{attribute 'GeneratedUsingTerminal: EK1122-0000-0018'}
{attribute addProperty BoxType "EK1122-0000-0018"}
{attribute addProperty Id "Beckhoff_EPP2xxxsub_EK1100EK1100_AB5A94672A_0001_EPP2008_0001_0016EPP2008_D86968E311A_0002_EPP2008_0001_0017EPP2008_D86968E311A_0003_EPP2008_0001_0018EPP2008_D86968E311A_0004_EPP2008_0002_0016EPP2008_D86968E311A_0005_EPP2008_0002_0017EPP2008_D86968E311A_0006_EPP2008_0002_0018EPP2008_D86968E311A_0007_EPP2008_0022_0016EPP2008_D86968E311A_0008_EPP2028_0001_0016EPP2028_D86968E311A_0009_EPP2028_0001_0017EPP2028_D86968E311A_0010_EPP2028_0002_0016EPP2028_D86968E311A_0011_EPP2028_0002_0017EPP2028_D86968E311A_0012_EPP2038_0001_0016EPP2038_0667821720A_0013_EPP2038_0002_0016EPP2038_0667821720A_0014_EPP2304_0061_0016EPP2304_2989DBB88A_0015_EPP2304_0061_0017EPP2304_2989DBB88A_0016_EPP2304_0061_0018EPP2304_2989DBB88A_0017_EPP2308_0001_0016EPP2308_CC30ABA712A_0018_EPP2308_0001_0017EPP2308_CC30ABA712A_0019_EPP2308_0001_0018EPP2308_CC30ABA712A_0020_EPP2308_0002_0016EPP2308_CC30ABA712A_0021_EPP2308_0002_0017EPP2308_CC30ABA712A_0022_EPP2308_0002_0018EPP2308_CC30ABA712A_0023_EPP2316_0003_0016EPP2316_ACB55CD744A_0024_EPP2316_0003_0017EPP2316_ACB55CD744A_0025_EPP2316_0003_0018EPP2316_B4F7513944A_0026_EPP2316_0008_0016EPP2316_ACB55CD744A_0027_EPP2316_0008_0017EPP2316_ACB55CD744A_0028_EPP2316_0008_0018EPP2316_B4F7513944A_0029_EPP2318_0001_0016EPP2318_CC30ABA712A_0030_EPP2318_0001_0017EPP2318_CC30ABA712A_0031_EPP2318_0001_0018EPP2318_CC30ABA712A_0032_EPP2318_0002_0016EPP2318_CC30ABA712A_0033_EPP2318_0002_0017EPP2318_CC30ABA712A_0034_EPP2318_0002_0018EPP2318_CC30ABA712A_0035_EPP2328_0001_0016EPP2328_CC30ABA712A_0036_EPP2328_0001_0017EPP2328_CC30ABA712A_0037_EPP2328_0001_0018EPP2328_CC30ABA712A_0038_EPP2328_0002_0016EPP2328_CC30ABA712A_0039_EPP2328_0002_0017EPP2328_CC30ABA712A_0040_EPP2328_0002_0018EPP2328_CC30ABA712A_0041_EPP2334_0061_0016EPP2334_CC30ABA712A_0042_EPP2334_0061_0017EPP2334_CC30ABA712A_0043_EPP2334_0061_0018EPP2334_CC30ABA712A_0044_EPP2334_0061_0019EPP2334_CC30ABA712A_0045_EPP2338_0001_0016EPP2338_B9F455E920A_0046_EPP2338_0001_0017EPP2338_B9F455E920A_0047_EPP2338_0001_0018EPP2338_B9F455E920A_0048_EPP2338_0002_0016EPP2338_B9F455E920A_0049_EPP2338_0002_0017EPP2338_B9F455E920A_0050_EPP2338_0002_0018EPP2338_B9F455E920A_0051_EPP2338_1001_0017EPP2338_B9F455E920A_0052_EPP2338_1001_0018EPP2338_B9F455E920A_0053_EPP2338_1001_0019EPP2338_B9F455E920A_0054_EPP2338_1002_0017EPP2338_B9F455E920A_0055_EPP2338_1002_0018EPP2338_B9F455E920A_0056_EPP2338_1002_0019EPP2338_B9F455E920A_0057_EPP2339_0003_0016EPP2339_509ECB0F50A_0058_EPP2339_0021_0016EPP2339_618EB00436A_0059_EPP2339_0021_0017EPP2339_0ADD710F36A_0060_EPP2339_0021_0018EPP2339_0ADD710F36A_0061_EPP2339_0022_0016EPP2339_618EB00436A_0062_EPP2339_0022_0017EPP2339_0ADD710F36A_0063_EPP2339_0022_0018EPP2339_0ADD710F36A_0064_EPP2349_0021_0016EPP2349_618EB00436A_0065_EPP2349_0021_0017EPP2349_0ADD710F36A_0066_EPP2349_0021_0018EPP2349_0ADD710F36A_0067_EPP2349_0022_0016EPP2349_618EB00436A_0068_EPP2349_0022_0017EPP2349_0ADD710F36A_0069_EPP2349_0022_0018EPP2349_0ADD710F36A_0070_EPP2624_0002_0016EPP2624_15DDA43F7A_0071_EPP2809_0021_0016EPP2809_E4096AA219A_0072_EPP2809_0022_0016EPP2809_E4096AA219A_0073_EPP2816_0004_0016EPP2816_C5A667B351A_0074_EPP2816_0004_0017EPP2816_C5A667B351A_0075_EPP2816_0008_0016EPP2816_2E3F94AC51A_0076_EPP2816_0008_0017EPP2816_2E3F94AC51A_0077_EPP2816_0008_0018EPP2816_2E3F94AC51A_0078_EPP2816_0010_0016EPP2816_2E3F94AC51A_0079_EPP2816_0010_0017EPP2816_2E3F94AC51A_0080_EPP2816_0010_0018EPP2816_2E3F94AC51A_0081_EPP2817_0008_0016EPP2817_1E85A59C70A_0082_EPP2817_0008_0017EPP2817_1E85A59C70A_0083_EPP2817_0008_0018EPP2817_1E85A59C70"}
{attribute addProperty CRC "1991220122"}
{attribute addProperty Size "2100"}
TYPE Beckhoff_EPP2xxxEK1122_76AF9B9A EXTENDS EK1122_AB5A9467 :
STRUCT
	{attribute addProperty Name "Beckhoff_EPP2xxxsub_EK1100"}
	Beckhoff_EPP2xxxsub_EK1100 : EK1100_AB5A9467;
	{attribute addProperty Name "A_0001_EPP2008_0001_0016"}
	A_0001_EPP2008_0001_0016 : EPP2008_D86968E3;
	{attribute addProperty Name "A_0002_EPP2008_0001_0017"}
	A_0002_EPP2008_0001_0017 : EPP2008_D86968E3;
	{attribute addProperty Name "A_0003_EPP2008_0001_0018"}
	A_0003_EPP2008_0001_0018 : EPP2008_D86968E3;
	{attribute addProperty Name "A_0004_EPP2008_0002_0016"}
	A_0004_EPP2008_0002_0016 : EPP2008_D86968E3;
	{attribute addProperty Name "A_0005_EPP2008_0002_0017"}
	A_0005_EPP2008_0002_0017 : EPP2008_D86968E3;
	{attribute addProperty Name "A_0006_EPP2008_0002_0018"}
	A_0006_EPP2008_0002_0018 : EPP2008_D86968E3;
	{attribute addProperty Name "A_0007_EPP2008_0022_0016"}
	A_0007_EPP2008_0022_0016 : EPP2008_D86968E3;
	{attribute addProperty Name "A_0008_EPP2028_0001_0016"}
	A_0008_EPP2028_0001_0016 : EPP2028_D86968E3;
	{attribute addProperty Name "A_0009_EPP2028_0001_0017"}
	A_0009_EPP2028_0001_0017 : EPP2028_D86968E3;
	{attribute addProperty Name "A_0010_EPP2028_0002_0016"}
	A_0010_EPP2028_0002_0016 : EPP2028_D86968E3;
	{attribute addProperty Name "A_0011_EPP2028_0002_0017"}
	A_0011_EPP2028_0002_0017 : EPP2028_D86968E3;
	{attribute addProperty Name "A_0012_EPP2038_0001_0016"}
	A_0012_EPP2038_0001_0016 : EPP2038_06678217;
	{attribute addProperty Name "A_0013_EPP2038_0002_0016"}
	A_0013_EPP2038_0002_0016 : EPP2038_06678217;
	{attribute addProperty Name "A_0014_EPP2304_0061_0016"}
	A_0014_EPP2304_0061_0016 : EPP2304_2989DBB8;
	{attribute addProperty Name "A_0015_EPP2304_0061_0017"}
	A_0015_EPP2304_0061_0017 : EPP2304_2989DBB8;
	{attribute addProperty Name "A_0016_EPP2304_0061_0018"}
	A_0016_EPP2304_0061_0018 : EPP2304_2989DBB8;
	{attribute addProperty Name "A_0017_EPP2308_0001_0016"}
	A_0017_EPP2308_0001_0016 : EPP2308_CC30ABA7;
	{attribute addProperty Name "A_0018_EPP2308_0001_0017"}
	A_0018_EPP2308_0001_0017 : EPP2308_CC30ABA7;
	{attribute addProperty Name "A_0019_EPP2308_0001_0018"}
	A_0019_EPP2308_0001_0018 : EPP2308_CC30ABA7;
	{attribute addProperty Name "A_0020_EPP2308_0002_0016"}
	A_0020_EPP2308_0002_0016 : EPP2308_CC30ABA7;
	{attribute addProperty Name "A_0021_EPP2308_0002_0017"}
	A_0021_EPP2308_0002_0017 : EPP2308_CC30ABA7;
	{attribute addProperty Name "A_0022_EPP2308_0002_0018"}
	A_0022_EPP2308_0002_0018 : EPP2308_CC30ABA7;
	{attribute addProperty Name "A_0023_EPP2316_0003_0016"}
	A_0023_EPP2316_0003_0016 : EPP2316_ACB55CD7;
	{attribute addProperty Name "A_0024_EPP2316_0003_0017"}
	A_0024_EPP2316_0003_0017 : EPP2316_ACB55CD7;
	{attribute addProperty Name "A_0025_EPP2316_0003_0018"}
	A_0025_EPP2316_0003_0018 : EPP2316_B4F75139;
	{attribute addProperty Name "A_0026_EPP2316_0008_0016"}
	A_0026_EPP2316_0008_0016 : EPP2316_ACB55CD7;
	{attribute addProperty Name "A_0027_EPP2316_0008_0017"}
	A_0027_EPP2316_0008_0017 : EPP2316_ACB55CD7;
	{attribute addProperty Name "A_0028_EPP2316_0008_0018"}
	A_0028_EPP2316_0008_0018 : EPP2316_B4F75139;
	{attribute addProperty Name "A_0029_EPP2318_0001_0016"}
	A_0029_EPP2318_0001_0016 : EPP2318_CC30ABA7;
	{attribute addProperty Name "A_0030_EPP2318_0001_0017"}
	A_0030_EPP2318_0001_0017 : EPP2318_CC30ABA7;
	{attribute addProperty Name "A_0031_EPP2318_0001_0018"}
	A_0031_EPP2318_0001_0018 : EPP2318_CC30ABA7;
	{attribute addProperty Name "A_0032_EPP2318_0002_0016"}
	A_0032_EPP2318_0002_0016 : EPP2318_CC30ABA7;
	{attribute addProperty Name "A_0033_EPP2318_0002_0017"}
	A_0033_EPP2318_0002_0017 : EPP2318_CC30ABA7;
	{attribute addProperty Name "A_0034_EPP2318_0002_0018"}
	A_0034_EPP2318_0002_0018 : EPP2318_CC30ABA7;
	{attribute addProperty Name "A_0035_EPP2328_0001_0016"}
	A_0035_EPP2328_0001_0016 : EPP2328_CC30ABA7;
	{attribute addProperty Name "A_0036_EPP2328_0001_0017"}
	A_0036_EPP2328_0001_0017 : EPP2328_CC30ABA7;
	{attribute addProperty Name "A_0037_EPP2328_0001_0018"}
	A_0037_EPP2328_0001_0018 : EPP2328_CC30ABA7;
	{attribute addProperty Name "A_0038_EPP2328_0002_0016"}
	A_0038_EPP2328_0002_0016 : EPP2328_CC30ABA7;
	{attribute addProperty Name "A_0039_EPP2328_0002_0017"}
	A_0039_EPP2328_0002_0017 : EPP2328_CC30ABA7;
	{attribute addProperty Name "A_0040_EPP2328_0002_0018"}
	A_0040_EPP2328_0002_0018 : EPP2328_CC30ABA7;
	{attribute addProperty Name "A_0041_EPP2334_0061_0016"}
	A_0041_EPP2334_0061_0016 : EPP2334_CC30ABA7;
	{attribute addProperty Name "A_0042_EPP2334_0061_0017"}
	A_0042_EPP2334_0061_0017 : EPP2334_CC30ABA7;
	{attribute addProperty Name "A_0043_EPP2334_0061_0018"}
	A_0043_EPP2334_0061_0018 : EPP2334_CC30ABA7;
	{attribute addProperty Name "A_0044_EPP2334_0061_0019"}
	A_0044_EPP2334_0061_0019 : EPP2334_CC30ABA7;
	{attribute addProperty Name "A_0045_EPP2338_0001_0016"}
	A_0045_EPP2338_0001_0016 : EPP2338_B9F455E9;
	{attribute addProperty Name "A_0046_EPP2338_0001_0017"}
	A_0046_EPP2338_0001_0017 : EPP2338_B9F455E9;
	{attribute addProperty Name "A_0047_EPP2338_0001_0018"}
	A_0047_EPP2338_0001_0018 : EPP2338_B9F455E9;
	{attribute addProperty Name "A_0048_EPP2338_0002_0016"}
	A_0048_EPP2338_0002_0016 : EPP2338_B9F455E9;
	{attribute addProperty Name "A_0049_EPP2338_0002_0017"}
	A_0049_EPP2338_0002_0017 : EPP2338_B9F455E9;
	{attribute addProperty Name "A_0050_EPP2338_0002_0018"}
	A_0050_EPP2338_0002_0018 : EPP2338_B9F455E9;
	{attribute addProperty Name "A_0051_EPP2338_1001_0017"}
	A_0051_EPP2338_1001_0017 : EPP2338_B9F455E9;
	{attribute addProperty Name "A_0052_EPP2338_1001_0018"}
	A_0052_EPP2338_1001_0018 : EPP2338_B9F455E9;
	{attribute addProperty Name "A_0053_EPP2338_1001_0019"}
	A_0053_EPP2338_1001_0019 : EPP2338_B9F455E9;
	{attribute addProperty Name "A_0054_EPP2338_1002_0017"}
	A_0054_EPP2338_1002_0017 : EPP2338_B9F455E9;
	{attribute addProperty Name "A_0055_EPP2338_1002_0018"}
	A_0055_EPP2338_1002_0018 : EPP2338_B9F455E9;
	{attribute addProperty Name "A_0056_EPP2338_1002_0019"}
	A_0056_EPP2338_1002_0019 : EPP2338_B9F455E9;
	{attribute addProperty Name "A_0057_EPP2339_0003_0016"}
	A_0057_EPP2339_0003_0016 : EPP2339_509ECB0F;
	{attribute addProperty Name "A_0058_EPP2339_0021_0016"}
	A_0058_EPP2339_0021_0016 : EPP2339_618EB004;
	{attribute addProperty Name "A_0059_EPP2339_0021_0017"}
	A_0059_EPP2339_0021_0017 : EPP2339_0ADD710F;
	{attribute addProperty Name "A_0060_EPP2339_0021_0018"}
	A_0060_EPP2339_0021_0018 : EPP2339_0ADD710F;
	{attribute addProperty Name "A_0061_EPP2339_0022_0016"}
	A_0061_EPP2339_0022_0016 : EPP2339_618EB004;
	{attribute addProperty Name "A_0062_EPP2339_0022_0017"}
	A_0062_EPP2339_0022_0017 : EPP2339_0ADD710F;
	{attribute addProperty Name "A_0063_EPP2339_0022_0018"}
	A_0063_EPP2339_0022_0018 : EPP2339_0ADD710F;
	{attribute addProperty Name "A_0064_EPP2349_0021_0016"}
	A_0064_EPP2349_0021_0016 : EPP2349_618EB004;
	{attribute addProperty Name "A_0065_EPP2349_0021_0017"}
	A_0065_EPP2349_0021_0017 : EPP2349_0ADD710F;
	{attribute addProperty Name "A_0066_EPP2349_0021_0018"}
	A_0066_EPP2349_0021_0018 : EPP2349_0ADD710F;
	{attribute addProperty Name "A_0067_EPP2349_0022_0016"}
	A_0067_EPP2349_0022_0016 : EPP2349_618EB004;
	{attribute addProperty Name "A_0068_EPP2349_0022_0017"}
	A_0068_EPP2349_0022_0017 : EPP2349_0ADD710F;
	{attribute addProperty Name "A_0069_EPP2349_0022_0018"}
	A_0069_EPP2349_0022_0018 : EPP2349_0ADD710F;
	{attribute addProperty Name "A_0070_EPP2624_0002_0016"}
	A_0070_EPP2624_0002_0016 : EPP2624_15DDA43F;
	{attribute addProperty Name "A_0071_EPP2809_0021_0016"}
	A_0071_EPP2809_0021_0016 : EPP2809_E4096AA2;
	{attribute addProperty Name "A_0072_EPP2809_0022_0016"}
	A_0072_EPP2809_0022_0016 : EPP2809_E4096AA2;
	{attribute addProperty Name "A_0073_EPP2816_0004_0016"}
	A_0073_EPP2816_0004_0016 : EPP2816_C5A667B3;
	{attribute addProperty Name "A_0074_EPP2816_0004_0017"}
	A_0074_EPP2816_0004_0017 : EPP2816_C5A667B3;
	{attribute addProperty Name "A_0075_EPP2816_0008_0016"}
	A_0075_EPP2816_0008_0016 : EPP2816_2E3F94AC;
	{attribute addProperty Name "A_0076_EPP2816_0008_0017"}
	A_0076_EPP2816_0008_0017 : EPP2816_2E3F94AC;
	{attribute addProperty Name "A_0077_EPP2816_0008_0018"}
	A_0077_EPP2816_0008_0018 : EPP2816_2E3F94AC;
	{attribute addProperty Name "A_0078_EPP2816_0010_0016"}
	A_0078_EPP2816_0010_0016 : EPP2816_2E3F94AC;
	{attribute addProperty Name "A_0079_EPP2816_0010_0017"}
	A_0079_EPP2816_0010_0017 : EPP2816_2E3F94AC;
	{attribute addProperty Name "A_0080_EPP2816_0010_0018"}
	A_0080_EPP2816_0010_0018 : EPP2816_2E3F94AC;
	{attribute addProperty Name "A_0081_EPP2817_0008_0016"}
	A_0081_EPP2817_0008_0016 : EPP2817_1E85A59C;
	{attribute addProperty Name "A_0082_EPP2817_0008_0017"}
	A_0082_EPP2817_0008_0017 : EPP2817_1E85A59C;
	{attribute addProperty Name "A_0083_EPP2817_0008_0018"}
	A_0083_EPP2817_0008_0018 : EPP2817_1E85A59C;
END_STRUCT
END_TYPE

(* stored: Version 1.2.0.0, ProductVersion 3.1.4024.9
   DUT Beckhoff_EPP2xxxEK1122_76AF9B9A: Id {35888cff-3890-48cb-998d-99614031967e} *)
